(* IEC 61131-3 sources: CodesysTest/export/UN00 - Sharp Bagger/EM01 - Bagger Head/EM01_BaggerHead.pou, 1 file *)

(* ---- EM01_BaggerHead.pou.st ---- *)
(*#-#-#-#-#-#-#-#-#-#---Declaration---#-#-#-#-#-#-#-#-#-#-#-#-#*)

FUNCTION_BLOCK EM01_BaggerHead EXTENDS FB_PackMLStates IMPLEMENTS IEM01_BaggerHead
VAR_INPUT
	(*Comnponents*)
	bagOpenFingers : IBagOpenFingers;
	sealFlatteners : ISealFlatteners;
	sealer : ISealer;
	pressureBar : IPressureBar;
	printer : IPrinter;
	bagDelivery : IBagDelivery;
	vacuumBagOpen : IVacuumBagOpen;
	IBD : I_IBD;
	barcodeVerifier : IBarcodeVerifier;
	{warning 'TODO: Move Load Plate to discharge, not baggerhead'}
	loadPlate : IRetractingLoadPlate;
	(*Options and settings*)
	bagOpenAssistEnabled : BOOL;		// Bag Open Assist Option Enabled from HMI
	bagOpenSensorEnabled : BOOL;		// Bag Open Sensors Enabled from HMI
	separateBeforeSealEnabled : BOOL;	// Separate before Seal Option Enabled from HMI
	bagOpenRetrySetting : UINT;
	newJobLoaded : BOOL;
	vacuumDwell : TIME;
	cancelPrint : BOOL;
END_VAR
VAR_OUTPUT
	bagOpenRetryCount : UINT;
	failedToOpenBag : FB_Fault(name := CONCAT(_prefix,'Failed to Open Bag'));
	barcodeVerificationFailed : FB_Fault(name := CONCAT(_prefix,'Barcode Fail'));
END_VAR
VAR
	_startCycle : BOOL;
	_readyToAcceptProduct : BOOL;
END_VAR
(*#-#-#-#-#-#-#-#-#-#---Implementation---#-#-#-#-#-#-#-#-#-#-#-#-#*)
